FUNCTION_BLOCK FB_DiagnosisEtherCATSlaveWc0 IMPLEMENTS I_DiagnosisEtherCATSlave
VAR_INPUT
	sSlaveName					:STRING	:='NameNotSet';				//スレーブ名
END_VAR
VAR
	_bError						:BOOL;
	
	fbStateDiagnosis			:FB_StateDiagnosis;
END_VAR

(*エラー発生を出力*)
PROPERTY bError : BOOL
GET
bError:=_bError;
END_GET
END_PROPERTY

(*呼び出して診断実行*)
METHOD Execute
//診断用FBを呼び出し
fbStateDiagnosis(sSlaveName:=sSlaveName);

_bError:=fbStateDiagnosis.bError;
END_METHOD

END_FUNCTION_BLOCK

(* stored: Version 1.1.0.1
   POU FB_DiagnosisEtherCATSlaveWc0: Id {519e11a6-b44d-418f-ae09-7534acbef856}, SpecialFunc None
   Property bError: Id {1c16415b-74b3-4c00-9639-b2d012b9e032}
   Get Get: Id {e0b87b6b-9e8d-4c58-a06f-6639d9afd085}
   Method Execute: Id {892d64d4-7ff8-47e0-acfa-e3ca66eeed7e} *)
